// TIA Portal V21 export
FUNCTION "Dodawanie" : Void   // FC2, LAD
{ S7_Optimized_Access := 'TRUE' }
// stored: SetENOAutomatically false
BEGIN

REGION Network 1
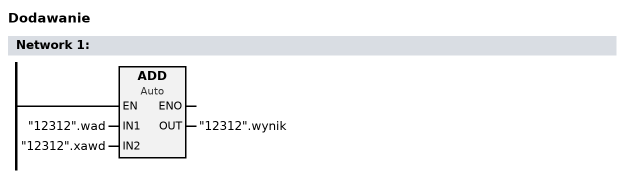
   RUNG wire#powerrail
      { S7_GenerateENO := "TRUE" } Add(in1 := "12312".wad, in2 := "12312".xawd, out => "12312".wynik)
   END_RUNG
   // the same network as SCL:
   "12312".wynik := "12312".wad + "12312".xawd;
END_REGION
END_FUNCTION
